// Mitsubishi GX Works2 project: 타이머 예제 1   PLC: Q03UDV

PROGRAM MAIN
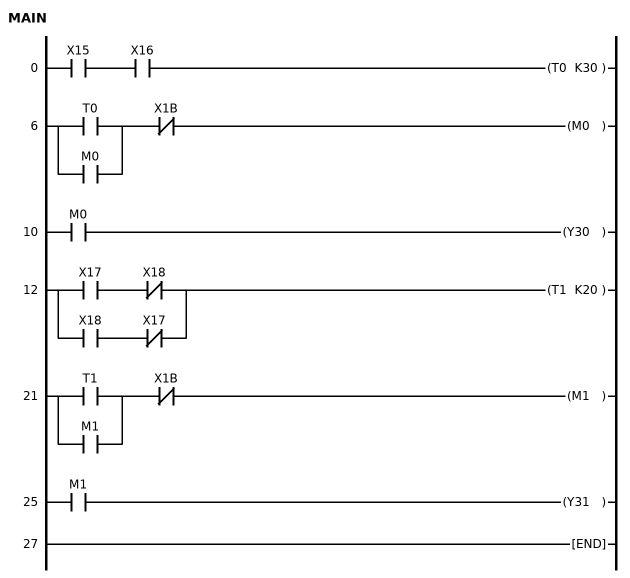
0     LD      X15
      AND     X16
      OUT     T0 K30
6     LD      T0
      OR      M0
      ANI     X1B
      OUT     M0
10    LD      M0
      OUT     Y30
12    LD      X17
      ANI     X18
      LD      X18
      ANI     X17
      ORB
      OUT     T1 K20
21    LD      T1
      OR      M1
      ANI     X1B
      OUT     M1
25    LD      M1
      OUT     Y31
27    END
END_PROGRAM
